TYPE Sfts_Instruction_DUT :
STRUCT
	Mode_Change:  UINT;
	Enable:  BOOL;
	Extend:  Bool;
	Retract:  Bool;
	Manual_Extend:  Bool;
	Manual_Retract:  BOOL;
END_STRUCT
END_TYPE

(* stored: Version 1.1.0.1
   DUT Sfts_Instruction_DUT: Id {12324132-49cb-4263-aa23-232df787f5ff} *)
